// Output from slave arm control task, including arm status and cartesian data
// Input to safety task and Master controller
TYPE ST_SlaveStatus :
STRUCT
	
	// state machine
	m_armState:ARRAY[1..g_sArmNum] OF E_SlaveArmState:=[g_sArmNum(SlaveArmState_Error)];
	
	// self-check pass flag
	m_selfCheckPass :ARRAY[1..g_sArmNum] OF BOOL :=[4(False)];
	
	// instrument info
	m_instruStauts :ARRAY[1..g_sArmNum] OF ST_InstruStatus;
	
	// flag if endoscope is mounted
	m_endoscopeMounted :BOOL := FALSE;
	
	// endoscope pose in cart coordinate
	m_endoscopePose : ST_Frame;
	
	// command arm pose in slave arm coordinate
	m_cmdArmPose:ARRAY[1..g_sArmNum] OF ST_Frame;
	
	// current arm pose in slave arm coordinate
	m_curArmPose:ARRAY[1..g_sArmNum] OF ST_Frame;
	
	// command arm twist[linear velocity; angular veloicty] in  slave arm coordinate
	m_cmdArmTwist:ARRAY[1..g_sArmNum] OF Vec6d;
	
	// current arm twist[linear velocity; angular veloicty] in  slave arm coordinate
	m_curArmTwist:ARRAY[1..g_sArmNum] OF vec6d;
	
	// master slave pose error [position, angle*axis] in endoscope coordinate
	m_masterSlavePoseError :ARRAY[1..g_sArmNum] OF Vec6d; 

END_STRUCT
END_TYPE

(* stored: Version 1.1.0.1, ProductVersion 3.1.4024.12
   DUT ST_SlaveStatus: Id {8673ecde-c145-4df2-8157-2e6da5d46538} *)
